// TIA Portal V20 export
TYPE "Station"
   STRUCT
      SensorA : Bool;
      SensorB : Bool;
      SensorC : Bool;
      SensorD : Bool;
      IsEmpty : Bool;
      IsOccupied : Bool;
      Numer : SInt;
      Row : SInt;
      Column : SInt;
   END_STRUCT;
END_TYPE
